Staubli VAL3: isActive.pgx

public program isActive(bool& x_bActive[], string x_sItem)
  local num l_nSize
begin
  // check if is active
  x_bActive=saveInOut:dOutput[x_sItem].bActive
end
